(*
SPDX-FileCopyrightText: © 2026 Oleksandr Tiutyk <trofimich@gmail.com>
SPDX-License-Identifier: MIT
License: https://opensource.org/license/mit
*)

(*!
<summary>Changes a value from a starting value to a target over a specified duration.</summary>
<description>
Start and Execute use the same cyclic task. Execute must be called once per task cycle; skipped calls are not
supported. An optional target reference is borrowed and must remain valid while used by the ramp. Each timer
step accumulates the task period in LTIME and calculates the output from the starting value. Completion
depends on accumulated duration, not floating-point equality. A zero duration completes immediately in Start.
</description>
*)

{attribute 'no_explicit_call' := 'do not call this function block directly'}
FUNCTION_BLOCK LinearRamp EXTENDS Object IMPLEMENTS IExecutable
VAR_STAT
	//! <summary>Class name shared by all instances of this function block.</summary>
	{attribute 'hide'} 
	_ClassName : STRING := __POUNAME();
END_VAR
VAR		
	{attribute 'hide'} 
	_StartValue : LREAL;
	{attribute 'hide'} 
	_EndValue : LREAL;
	{attribute 'hide'} 
	_TransitionTime : TIME;
	
	{attribute 'hide'} 
	_LocalCurrentValue : LREAL;
	{attribute 'hide'} 
	_CurrentValueReference : REFERENCE TO LREAL REF= _LocalCurrentValue;
	{attribute 'hide'} 
	_RemainingTime : TIME;
	
	{attribute 'hide'} 
	_ElapsedTime : LTIME;
	
	{attribute 'hide'} 
	_Timer : Tc2_Standard.LTON;
END_VAR

(*!
<summary>Reports that a transition timer is active and not complete.</summary>
<description>Read-only view of the most recent Start/Execute state; reading does not advance the ramp.</description>
*)
{attribute 'monitoring' := 'call'}
PROPERTY FINAL Busy : BOOL
GET
Busy := _Timer.IN AND_THEN NOT _Timer.Q;
END_GET
END_PROPERTY

{attribute 'monitoring' := 'call'}
PROPERTY ClassName : REFERENCE TO STRING
GET
ClassName REF= _ClassName;
END_GET
END_PROPERTY

(*!
<summary>Reads the current ramp target storage.</summary>
<description>
Returns the value through the active internal or borrowed reference. The external reference, when supplied to
Start, must remain alive; reading does not advance the transition.
</description>
*)
{attribute 'monitoring' := 'call'}
PROPERTY FINAL CurrentValue : LREAL
GET
CurrentValue := _CurrentValueReference;
END_GET
END_PROPERTY

(*!
<summary>Reports completion indicated by the ramp timer.</summary>
<description>Read-only view; updates follow Start/Execute and reading does not advance the ramp.</description>
*)
{attribute 'monitoring' := 'call'}
PROPERTY FINAL Done : BOOL
GET
Done := _Timer.Q;
END_GET
END_PROPERTY

(*!
<summary>Returns the target value recorded for the latest transition.</summary>
<description>Read-only snapshot set by Start.</description>
*)
{attribute 'monitoring' := 'call'}
PROPERTY FINAL EndValue : LREAL
GET
EndValue := _EndValue;
END_GET
END_PROPERTY

(*!
<summary>Advances the transition by one step when the task-period timer expires.</summary>
<description>
Call once per cycle in the same task as Start. Calls while not busy do nothing. Each expired timer adds one
task period to elapsed time and interpolates from the starting value. Once the accumulated time reaches the
duration, the transition writes the exact target value and clears RemainingTime. External writes to the
borrowed output do not change the interpolation.
</description>
*)
METHOD FINAL Execute
IF NOT Busy THEN
	RETURN;
END_IF

_Timer();

IF _Timer.Q THEN
	_ElapsedTime := _ElapsedTime + _Timer.PT;

	IF _ElapsedTime < TO_LTIME(_TransitionTime) THEN
		_CurrentValueReference := _StartValue + (_EndValue - _StartValue)
			* (TO_LREAL(TO_ULINT(_ElapsedTime)) / TO_LREAL(TO_ULINT(TO_LTIME(_TransitionTime))));
		_RemainingTime := TO_TIME(TO_LTIME(_TransitionTime) - _ElapsedTime);

		_Timer(IN := FALSE);
		_Timer(IN := TRUE);
	ELSE
		_CurrentValueReference := _EndValue;
		_RemainingTime := Times.MIN_VALUE;
	END_IF
END_IF
END_METHOD

(*!
<summary>Provides the library namespace used in diagnostics.</summary>
<description>
Borrowed read-only reference to the compiler-initialized library namespace; no ownership transfer.
</description>
*)
{attribute 'monitoring' := 'call'}
PROPERTY NamespaceName : REFERENCE TO STRING
GET
NamespaceName REF= CurrentNamespace.Name;
END_GET
END_PROPERTY

(*!
<summary>Returns the cached remaining transition duration.</summary>
<description>
TIME has millisecond resolution. Reading does not advance Execute or the task-period-based progression.
</description>
*)
{attribute 'monitoring' := 'call'}
PROPERTY FINAL RemainingTime : TIME
GET
RemainingTime := _RemainingTime;
END_GET
END_PROPERTY

(*!
<summary>Reports the byte size of this concrete instance.</summary>
<description>
Uses XSIZEOF on the instance. Does not include separately allocated payloads or prove that an arbitrary
address is valid.
</description>
*)
{attribute 'monitoring' := 'call'}
PROPERTY SelfSize : ULINT
GET
SelfSize := XSIZEOF(THIS^);
END_GET
END_PROPERTY

(*!
<summary>Starts a transition from startValue to endValue.</summary>
<description>
Call from the cyclic task that will execute the ramp. A zero transitionTime immediately writes endValue,
clears RemainingTime, sets Done and clears Busy, including when replacing an active transition.
</description>
<param name="startValue">Initial value written when starting the transition.</param>
<param name="endValue">Target value of the transition.</param>
<param name="transitionTime">Requested duration; zero completes immediately.</param>
<param name="targetVariable">Optional borrowed output reference. When omitted, the ramp uses its internal value.</param>
*)
METHOD FINAL Start
VAR_INPUT
	startValue : LREAL;
	endValue : LREAL;
	transitionTime : TIME;
	targetVariable : REFERENCE TO LREAL := 0;
END_VAR
VAR
	plcTaskSystemInfo : Global.PlcTaskSystemInfo;
END_VAR
plcTaskSystemInfo := Tc2_System.F_GetTaskInfo();
	
_StartValue := startValue;
_EndValue := endValue;
_TransitionTime := transitionTime;

IF __ISVALIDREF(targetVariable) THEN
	_CurrentValueReference REF= targetVariable;
ELSE
	_CurrentValueReference REF= _LocalCurrentValue;
END_IF

_CurrentValueReference := startValue;
_RemainingTime := transitionTime;
_ElapsedTime := LongTimes.MIN_VALUE;

IF transitionTime > Times.MIN_VALUE THEN
	_Timer(IN := FALSE);
	_Timer(IN := TRUE, PT := TO_LTIME(TO_ULINT(plcTaskSystemInfo.CycleTime) * 100));
ELSE
	_CurrentValueReference := endValue;

	_Timer(IN := FALSE);
	_Timer(IN := TRUE, PT := LongTimes.MIN_VALUE);
END_IF
END_METHOD

(*!
<summary>Returns the starting value recorded for the latest transition.</summary>
<description>Read-only snapshot set by Start.</description>
*)
{attribute 'monitoring' := 'call'}
PROPERTY FINAL StartValue : LREAL
GET
StartValue := _StartValue;
END_GET
END_PROPERTY

(*!
<summary>Returns the requested transition duration.</summary>
<description>Read-only snapshot of the latest Start configuration, not elapsed time.</description>
*)
{attribute 'monitoring' := 'call'}
PROPERTY FINAL TransitionTime : TIME
GET
TransitionTime := _TransitionTime;
END_GET
END_PROPERTY

END_FUNCTION_BLOCK

(* stored: Version 1.1.0.1
   POU LinearRamp: Id {89e8744a-f710-43bd-a568-d953e4a14052}, SpecialFunc None
   Property Busy: Id {e507dedb-0cef-4d37-a7ad-b8295e5a074c}
   Get Get: Id {a5f784a9-fa56-4b25-9137-66072e50b328}
   Property ClassName: Id {7c4d8006-4a00-4f05-be1a-ab0d01b6a996}
   Get Get: Id {e087e48f-4d09-4681-9510-feb522f5ea2f}
   Property CurrentValue: Id {387a21ac-5037-4ea4-b4fa-aed89bced2be}
   Get Get: Id {f5bcde31-560e-406e-95c6-40cc3db71638}
   Property Done: Id {b15600da-2ee7-4fac-b194-aa237146bd58}
   Get Get: Id {8850af1b-66d0-407b-bc8e-312531041b44}
   Property EndValue: Id {89d139df-acd8-440b-bf9c-16efec2879af}
   Get Get: Id {f1cd132b-11d0-41ed-955f-6acb8a759a4b}
   Method Execute: Id {38af6e39-2e6c-4584-b59a-f0ec5df5767e}
   Property NamespaceName: Id {51b3e739-b297-40a9-8041-305d1afae442}
   Get Get: Id {626e1991-34f2-4cf8-8edb-9556d7cdb1c5}
   Property RemainingTime: Id {779cd677-5d00-40c9-8275-5fb992d1f419}
   Get Get: Id {b98c3ec4-ba18-40c2-a93c-4ad402a8bd7c}
   Property SelfSize: Id {eb227785-7431-4143-b5a9-32053381bc10}
   Get Get: Id {7f5ff5ad-e806-4cdc-b44e-30a1f978d9ff}
   Method Start: Id {a5b0c418-0d21-4c1d-83ea-0c355bceaebe}
   Property StartValue: Id {023a42a4-02cc-4e65-8dde-df189de525f0}
   Get Get: Id {708a4576-bab2-4bf8-9916-06aa289e79af}
   Property TransitionTime: Id {e4e1a5d8-7540-4b54-a217-e0ff4b16aefd}
   Get Get: Id {6de9dccc-dcc0-466a-aa5a-fe37372cab0e} *)
